FUNCTION_BLOCK VALFORMAT_1942D31DAE3706DC9 (* MBus device interface function block type *)
  (* Standard: 61499-2 *)
  (* Version 1.0, 09.09.2008, oberwal, nxtControl GmbH, Initial Version *)
  PACKAGE UAO.Hackathon;
  (* Compiler Cpp *)
  {SET_ATTRIBUTE(Runtime.FBType.ImplementingType, Runtime.Standard#DYNGEN_VALFORMAT)}
  {SET_ATTRIBUTE(Configuration.GenericFBType.InterfaceParams, Runtime.Standard#I:=3;VALUE${I$}:STRING,STRING,STRING)}
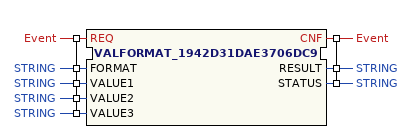
  EVENT_INPUT
    REQ WITH FORMAT, VALUE1, VALUE2, VALUE3; (* Request a formatting operation *)
  END_EVENT
  EVENT_OUTPUT
    CNF WITH RESULT, STATUS; (* Confirms a formattiong operation *)
  END_EVENT
  VAR_INPUT
    FORMAT : STRING; (* Defines a standard C printf like format *)
    VALUE1 : STRING; (* A list of values to be converted into a string as defined in parameter FORMAT *)
    VALUE2 : STRING; (* A list of values to be converted into a string as defined in parameter FORMAT *)
    VALUE3 : STRING; (* A list of values to be converted into a string as defined in parameter FORMAT *)
  END_VAR
  VAR_OUTPUT
    RESULT : STRING; (* The formatted result string *)
    STATUS : STRING; (* Error information *)
  END_VAR
  EC_STATES
    START;
  END_STATES
END_FUNCTION_BLOCK
